{attribute addProperty BoxType "ELM2642-0000-0016"}
{attribute addProperty Id "Y1BIT10.1251Y2BIT10.1252Y3BIT10.1253Y4BIT10.1254"}
{attribute addProperty CRC "3875429920"}
{attribute addProperty SizeInBites "16"}
{attribute addProperty SizeInBytes "2"}
TYPE Outputs_Channel_E6FE5E20 :
STRUCT
	{attribute addProperty Name "Y1"}
	Y1 : BIT;
	{attribute addProperty Name "Y2"}
	Y2 : BIT;
	{attribute addProperty Name "Y3"}
	Y3 : BIT;
	{attribute addProperty Name "Y4"}
	Y4 : BIT;
	{attribute 'hide'}
	reserve_1_BIT_0 : BIT;
	{attribute 'hide'}
	reserve_1_BIT_1 : BIT;
	{attribute 'hide'}
	reserve_1_BIT_2 : BIT;
	{attribute 'hide'}
	reserve_1_BIT_3 : BIT;
	{attribute 'hide'}
	reserve_1_BIT_4 : BIT;
	{attribute 'hide'}
	reserve_1_BIT_5 : BIT;
	{attribute 'hide'}
	reserve_1_BIT_6 : BIT;
	{attribute 'hide'}
	reserve_1_BIT_7 : BIT;
	{attribute 'hide'}
	reserve_1_BIT_8 : BIT;
	{attribute 'hide'}
	reserve_1_BIT_9 : BIT;
	{attribute 'hide'}
	reserve_1_BIT_10 : BIT;
	{attribute 'hide'}
	reserve_1_BIT_11 : BIT;
END_STRUCT
END_TYPE

(* stored: Version 1.2.0.0, ProductVersion 3.1.4024.9
   DUT Outputs_Channel_E6FE5E20: Id {9c807486-5563-4289-9482-a55ecc58acfb} *)
